(* IEC 61131-3 sources: nvidia-ai-factory-controls/projects/IPC-02_Cooling/GVLs, 2 files *)

(* ---- GVL_CrossTask.gvl ---- *)
(* =============================================================================
    GVL_CrossTask — Cross-Task Data Exchange Buffer
    IPC-02: Cooling Control | NVIDIA AI Factory Controls
   =============================================================================

   PURPOSE:
     Provides the ONLY mechanism for data exchange between tasks.
     Prevents race conditions by enforcing atomic struct copy pattern.

   ARCHITECTURE:
     ┌─────────────────┐         ┌──────────────────────┐
     │  Control_Task   │         │  Communication_Task  │
     │  (5ms cycle)    │         │  (100ms cycle)       │
     │                 │         │                      │
     │  FB_CDU writes  │──copy──→│  Reads stCDU_Status  │──→ OPC UA
     │  stCDU_Status   │         │  at start of cycle   │
     │  at end of scan │         │                      │
     │                 │         │  Writes stCDU_Config  │
     │  Reads config   │←─copy──│  (from OPC UA params) │
     │  at start of    │         │  at end of cycle     │
     │  scan           │         │                      │
     └─────────────────┘         └──────────────────────┘

   RULES:
     1. Control_Task WRITES status structs, READS config structs.
     2. Communication_Task READS status structs, WRITES config structs.
     3. Each task copies the ENTIRE struct at its cycle boundary.
     4. No field-by-field access across tasks — always full struct copy.
     5. CODESYS guarantees non-preemption within a task cycle, so
        a struct copy within one scan is atomic from other tasks' view.

   RACE CONDITION ANALYSIS:
     Q: Can Communication_Task read a half-written status struct?
     A: No. Control_Task writes the struct in one scan (5ms). The
        Communication_Task reads at its own cycle start (100ms).
        CODESYS task scheduling ensures tasks don't interrupt each other
        mid-cycle on single-core. On multi-core, use {attribute 'atomic'}
        or explicit semaphores (not needed here — single-core IPC).

   MULTI-CORE NOTE:
     If deploying on multi-core IPC (e.g., CX5240 with core isolation),
     add {attribute 'atomic'} to each variable, or use CODESYS
     SysSem library for explicit locking. Current design assumes
     single-core execution with cooperative task scheduling.
   ============================================================================= *)

{attribute 'qualified_only'}
VAR_GLOBAL
    (* ─── Control → Communication (status snapshots) ─── *)

    (* CDU status: written by Control_Task, read by Communication_Task *)
    stCDU_01_Status      : ST_CDU_Status;
    stCDU_02_Status      : ST_CDU_Status;
    stCDU_03_Status      : ST_CDU_Status;
    stCDU_04_Status      : ST_CDU_Status;

    (* ─── Communication → Control (configuration/commands) ─── *)

    (* CDU config: written by Communication_Task (OPC UA), read by Control_Task *)
    stCDU_01_Config      : ST_CDU_Config;
    stCDU_02_Config      : ST_CDU_Config;
    stCDU_03_Config      : ST_CDU_Config;
    stCDU_04_Config      : ST_CDU_Config;

    (* GPU telemetry: written by Communication_Task, read by Control_Task *)
    fGPU_Row1_TotalPower : REAL;    (* Total GPU power Row 1 [kW] *)
    fGPU_Row1_MaxTemp    : REAL;    (* Max GPU temp Row 1 [°C] *)
    fGPU_Row2_TotalPower : REAL;    (* Total GPU power Row 2 [kW] *)
    fGPU_Row2_MaxTemp    : REAL;    (* Max GPU temp Row 2 [°C] *)
    bGPU_DataFresh       : BOOL;    (* TRUE = GPU data updated within last 5s *)
    nGPU_UpdateCounter   : UDINT;   (* Increments on each GPU data update *)

    (* ─── Safety → All Tasks (safety permit) ─── *)

    (* Written by Safety_Task, read by all other tasks.
       Single BOOL — atomically readable on all architectures. *)
    bSafetyPermit_Global : BOOL := TRUE;
    bEmergencyStop_Global: BOOL := FALSE;
END_VAR

(* ---- GVL_OPCUA_Publish.gvl ---- *)
(* =============================================================================
    GVL_OPCUA_Publish — OPC UA Exposed Variables
    IPC-02: Cooling Control | NVIDIA AI Factory Controls
   =============================================================================

   PURPOSE:
     All variables in this GVL are exposed to the OPC UA server via
     CODESYS symbol configuration. External clients (edge gateway,
     SCADA, digital twin) read/write these variables.

   HOW IT WORKS:
     1. Communication_Task copies data FROM GVL_CrossTask INTO this GVL
     2. OPC UA server reads these variables (asynchronous, on client request)
     3. OPC UA clients write setpoints/commands to VAR_CONFIG section
     4. Communication_Task copies commands FROM this GVL TO GVL_CrossTask

   NAMING CONVENTION:
     Variable names here become OPC UA browse names.
     Hierarchy is created by the '.' separator in the variable name.
     Example: Cooling_CDU_01_SupplyTemp → OPC UA node: Cooling/CDU_01/SupplyTemp

   SYMBOL CONFIG:
     In CODESYS: Project → Symbol Configuration → Add GVL_OPCUA_Publish
     Set access: Read for status, ReadWrite for setpoints/commands.

   SECURITY:
     Setpoints and commands are in a separate section with explicit
     'readwrite' access. Status variables are read-only.
   ============================================================================= *)

{attribute 'symbol' := 'read'}
{attribute 'qualified_only'}
VAR_GLOBAL
    (* ═══════════════════════════════════════════════════════════════════════
       COOLING SYSTEM — Read-Only Status
       ═══════════════════════════════════════════════════════════════════════ *)

    (* --- CDU 01 --- *)
    Cooling_CDU_01_State         : USINT;       (* E_CDU_State as integer *)
    Cooling_CDU_01_Mode          : USINT;       (* E_CDU_Mode as integer *)
    Cooling_CDU_01_Healthy       : BOOL;
    Cooling_CDU_01_SupplyTemp    : REAL;        (* [°C] *)
    Cooling_CDU_01_ReturnTemp    : REAL;        (* [°C] *)
    Cooling_CDU_01_DeltaT        : REAL;        (* [°C] *)
    Cooling_CDU_01_FlowRate      : REAL;        (* [LPM] *)
    Cooling_CDU_01_Pressure      : REAL;        (* [bar] *)
    Cooling_CDU_01_PumpSpeed     : REAL;        (* [%] *)
    Cooling_CDU_01_ValvePos      : REAL;        (* [%] *)
    Cooling_CDU_01_Capacity_kW   : REAL;        (* [kW] *)
    Cooling_CDU_01_PumpRunning   : BOOL;
    Cooling_CDU_01_AtCapacity    : BOOL;
    Cooling_CDU_01_RunHours      : UDINT;       (* [hours] *)
    Cooling_CDU_01_StartCount    : UDINT;

    (* --- CDU 01 Alarms --- *)
    Cooling_CDU_01_Alm_TempHigh  : BOOL;
    Cooling_CDU_01_Alm_FlowLow  : BOOL;
    Cooling_CDU_01_Alm_Leak      : BOOL;
    Cooling_CDU_01_Alm_PumpFault : BOOL;
    Cooling_CDU_01_Alm_Pressure  : BOOL;
    Cooling_CDU_01_Alm_GPUWarn   : BOOL;

    (* --- CDU 02 (same structure) --- *)
    Cooling_CDU_02_State         : USINT;
    Cooling_CDU_02_Mode          : USINT;
    Cooling_CDU_02_Healthy       : BOOL;
    Cooling_CDU_02_SupplyTemp    : REAL;
    Cooling_CDU_02_ReturnTemp    : REAL;
    Cooling_CDU_02_DeltaT        : REAL;
    Cooling_CDU_02_FlowRate      : REAL;
    Cooling_CDU_02_Pressure      : REAL;
    Cooling_CDU_02_PumpSpeed     : REAL;
    Cooling_CDU_02_ValvePos      : REAL;
    Cooling_CDU_02_Capacity_kW   : REAL;
    Cooling_CDU_02_PumpRunning   : BOOL;
    Cooling_CDU_02_AtCapacity    : BOOL;

    (* --- System Totals --- *)
    Cooling_TotalCapacity_kW     : REAL;        (* Sum of all CDU capacity *)
    Cooling_FreeCoolingActive    : BOOL;        (* Economizer mode active *)
    Cooling_GPU_MaxTemp          : REAL;        (* Highest GPU temp across all zones [°C] *)
    Cooling_GPU_TotalPower_kW    : REAL;        (* Total GPU power [kW] *)

    (* ═══════════════════════════════════════════════════════════════════════
       SAFETY SYSTEM — Read-Only Status
       ═══════════════════════════════════════════════════════════════════════ *)
    Safety_SystemArmed           : BOOL;
    Safety_AnyZoneTripped        : BOOL;
    Safety_TrippedZoneCount      : USINT;
    Safety_InputFault            : BOOL;
    Safety_Permit                : BOOL;

    (* ═══════════════════════════════════════════════════════════════════════
       SYSTEM DIAGNOSTICS — Read-Only
       ═══════════════════════════════════════════════════════════════════════ *)
    System_Heartbeat_Control     : UDINT;       (* Control_Task heartbeat *)
    System_Heartbeat_Comm        : UDINT;       (* Communication_Task heartbeat *)
    System_Heartbeat_Safety      : UDINT;       (* Safety_Task heartbeat *)
    System_PublishRate_Hz        : REAL;         (* Actual publish rate *)
    System_PublishErrors         : UDINT;       (* Cumulative publish errors *)
    System_ActivePublishers      : USINT;       (* Connected publisher count *)
END_VAR

{attribute 'symbol' := 'readwrite'}
VAR_GLOBAL
    (* ═══════════════════════════════════════════════════════════════════════
       SETPOINTS & COMMANDS — Read-Write (from SCADA/cloud)
       ═══════════════════════════════════════════════════════════════════════ *)

    (* --- CDU Setpoints (operator adjustable) --- *)
    Cmd_CDU_01_SupplyTempSP      : REAL := 35.0;    (* Supply temp setpoint [°C] *)
    Cmd_CDU_01_Enable            : BOOL := TRUE;     (* CDU enable command *)
    Cmd_CDU_01_Mode              : USINT := 0;       (* Requested mode *)
    Cmd_CDU_01_ManualMode        : BOOL := FALSE;    (* Manual override *)
    Cmd_CDU_01_ManualPumpSpeed   : REAL := 0.0;      (* Manual pump [%] *)
    Cmd_CDU_01_ManualValvePos    : REAL := 0.0;      (* Manual valve [%] *)

    Cmd_CDU_02_SupplyTempSP      : REAL := 35.0;
    Cmd_CDU_02_Enable            : BOOL := TRUE;
    Cmd_CDU_02_Mode              : USINT := 0;

    (* --- System Commands --- *)
    Cmd_System_Reset             : BOOL := FALSE;    (* Global fault reset *)
    Cmd_EmergencyCool            : BOOL := FALSE;    (* Force all CDUs to MAX_COOL *)
END_VAR
